// TIA Portal V18 export
DATA_BLOCK "Data_block_1"   // DB1
{ S7_Optimized_Access := 'TRUE' }
// stored: MemoryReserve 100
   VAR
      var : Bool;
   END_VAR
BEGIN
END_DATA_BLOCK
